// TIA Portal project "Palletizer" (V17)

(* hardware
DEVICE "S71500/ET200MP-Station_1"  S7-1500 station
   slot 0: "Profilschiene_0"  6ES7 590-1***0-0AA0
   slot 1: "PLC_1"  CPU 1511-1 PN  6ES7 511-1AK00-0AB0  V1.8
   slot 2: "AI 8xU/I/RTD/TC ST_1"  AI 8xU/I/RTD/TC ST  6ES7 531-7KF00-0AB0  V2.0
   slot 3: "AI 8xU/I/RTD/TC ST_2"  AI 8xU/I/RTD/TC ST  6ES7 531-7KF00-0AB0  V2.0
   slot 4: "AI 8xU/I/RTD/TC ST_3"  AI 8xU/I/RTD/TC ST  6ES7 531-7KF00-0AB0  V2.0
   slot 5: "AI 8xU/I/RTD/TC ST_4"  AI 8xU/I/RTD/TC ST  6ES7 531-7KF00-0AB0  V2.0
   slot 6: "DI 16x24VDC BA_1"  DI 16x24VDC BA  6ES7 521-1BH10-0AA0  V1.0
*)

// ===== PLC "PLC_1"  CPU 1511-1 PN =====

VAR_GLOBAL   // PLC tag table "Standard-Variablentabelle"
   "PALLET AT ENTRY" AT %E0.0 : Bool;
   "pallet at exit" AT %I0.1 : Bool;
   "pallet loaded" AT %I0.2 : Bool;
   "box at entry" AT %I0.3 : Bool;
   "pusher limit" AT %I0.4 : Bool;
   "plate limit" AT %I0.5 : Bool;
   "clamped" AT %I0.6 : Bool;
   "elevator moving" AT %I0.7 : Bool;
   "start" AT %I1.0 : Bool;
   "reset" AT %I1.1 : Bool;
   "stop" AT %I1.2 : Bool;
   "emergency stop" AT %I1.3 : Bool;
   "auto" AT %I1.4 : Bool;
   "factory run" AT %I1.5 : Bool;
   "pallet feeder" AT %Q0.0 : Bool;
   "load pallet" AT %Q0.1 : Bool;
   "exit conveyor" AT %Q0.2 : Bool;
   "move to limit" AT %Q0.3 : Bool;
   "elevator up" AT %Q0.4 : Bool;
   "elevator down" AT %Q0.5 : Bool;
   "box feeder" AT %Q0.6 : Bool;
   "turn" AT %Q0.7 : Bool;
   "push" AT %Q1.0 : Bool;
   "load belt" AT %Q1.1 : Bool;
   "clamp" AT %Q1.2 : Bool;
   "open plate" AT %Q1.3 : Bool;
   "warning light" AT %Q1.4 : Bool;
   "start light" AT %Q1.5 : Bool;
   "reset light" AT %Q1.6 : Bool;
   "stop light" AT %Q1.7 : Bool;
   "Tag_1" AT %M0.0 : Bool;
   "Tag_2" AT %M0.1 : Bool;
   "Tag_3" AT %M0.2 : Bool;
   "Tag_4" AT %M0.3 : Bool;
   "Tag_5" AT %M0.4 : Bool;
   "Tag_6" AT %M0.6 : Bool;
   "Tag_7" AT %M1.0 : Bool;
   "Tag_8" AT %MD100 : Time;
   "Tag_9" AT %M1.1 : Bool;
   "Tag_10" AT %MW100 : Int;
   "Tag_11" AT %M1.2 : Bool;
   "Tag_12" AT %M1.3 : Bool;
   "Tag_13" AT %MD200 : Time;
   "Tag_14" AT %M1.4 : Bool;
   "Tag_15" AT %M1.5 : Bool;
   "Tag_16" AT %MD300 : Time;
   "Tag_17" AT %M2.1 : Bool;
   "Tag_18" AT %M2.3 : Bool;
   "Tag_19" AT %M3.2 : Bool;
   "Tag_20" AT %M5.4 : Bool;
   "Tag_21" AT %M5.5 : Bool;
   "Tag_22" AT %M6.4 : Bool;
   "Tag_23" AT %M6.1 : Bool;
   "Tag_24" AT %M7.1 : Bool;
   "Tag_25" AT %M6.6 : Bool;
   "Tag_26" AT %M7.2 : Bool;
   "Tag_27" AT %M7.3 : Bool;
   "Tag_28" AT %M1.7 : Bool;
   "Tag_29" AT %M2.2 : Bool;
   "Tag_30" AT %M5.6 : Bool;
   "Tag_31" AT %M7.6 : Bool;
   "Tag_32" AT %M8.1 : Bool;
   "Tag_33" AT %M2.4 : Bool;
   "Tag_34" AT %M2.5 : Bool;
   "Tag_35" AT %M2.6 : Bool;
   "Tag_36" AT %M10.1 : Bool;
   "Tag_37" AT %MW400 : Int;
   "Tag_38" AT %QD30 : DWord;
END_VAR

// folder: System blocks/Program resources

DATA_BLOCK "IEC_Counter_0_DB"   // DB1
{ S7_Optimized_Access := 'TRUE' }
AUTHOR : Simatic
FAMILY : IEC
NAME : CNTR
VERSION : 1.0
// stored: InstanceOfName IEC_COUNTER
"IEC_COUNTER"
BEGIN
END_DATA_BLOCK

DATA_BLOCK "IEC_Timer_0_DB_1"   // DB2
{ S7_Optimized_Access := 'TRUE' }
AUTHOR : Simatic
FAMILY : IEC
NAME : IEC_TMR
VERSION : 1.0
// stored: InstanceOfName IEC_TIMER
"IEC_TIMER"
BEGIN
END_DATA_BLOCK

DATA_BLOCK "IEC_Timer_0_DB"   // DB3
{ S7_Optimized_Access := 'TRUE' }
AUTHOR : Simatic
FAMILY : IEC
NAME : IEC_TMR
VERSION : 1.0
// stored: InstanceOfName IEC_TIMER
"IEC_TIMER"
BEGIN
END_DATA_BLOCK

DATA_BLOCK "IEC_Counter_0_DB_1"   // DB4
{ S7_Optimized_Access := 'TRUE' }
AUTHOR : Simatic
FAMILY : IEC
NAME : CNTR
VERSION : 1.0
// stored: InstanceOfName IEC_COUNTER
"IEC_COUNTER"
BEGIN
END_DATA_BLOCK

DATA_BLOCK "IEC_Timer_0_DB_2"   // DB5
{ S7_Optimized_Access := 'TRUE' }
AUTHOR : Simatic
FAMILY : IEC
NAME : IEC_TMR
VERSION : 1.0
// stored: InstanceOfName IEC_TIMER
"IEC_TIMER"
BEGIN
END_DATA_BLOCK

DATA_BLOCK "IEC_Timer_0_DB_3"   // DB6
{ S7_Optimized_Access := 'TRUE' }
AUTHOR : Simatic
FAMILY : IEC
NAME : IEC_TMR
VERSION : 1.0
// stored: InstanceOfName IEC_TIMER
"IEC_TIMER"
BEGIN
END_DATA_BLOCK

DATA_BLOCK "IEC_Timer_0_DB_4"   // DB7
{ S7_Optimized_Access := 'TRUE' }
AUTHOR : Simatic
FAMILY : IEC
NAME : IEC_TMR
VERSION : 1.0
// stored: InstanceOfName IEC_TIMER
"IEC_TIMER"
BEGIN
END_DATA_BLOCK

DATA_BLOCK "IEC_Counter_0_DB_2"   // DB8
{ S7_Optimized_Access := 'TRUE' }
AUTHOR : Simatic
FAMILY : IEC
NAME : CNTR
VERSION : 1.0
// stored: InstanceOfName IEC_COUNTER
"IEC_COUNTER"
BEGIN
END_DATA_BLOCK

DATA_BLOCK "IEC_Timer_0_DB_5"   // DB9
{ S7_Optimized_Access := 'TRUE' }
AUTHOR : Simatic
FAMILY : IEC
NAME : IEC_TMR
VERSION : 1.0
// stored: InstanceOfName IEC_TIMER
"IEC_TIMER"
BEGIN
END_DATA_BLOCK

DATA_BLOCK "IEC_Timer_0_DB_6"   // DB10
{ S7_Optimized_Access := 'TRUE' }
AUTHOR : Simatic
FAMILY : IEC
NAME : IEC_TMR
VERSION : 1.0
// stored: InstanceOfName IEC_TIMER
"IEC_TIMER"
BEGIN
END_DATA_BLOCK

DATA_BLOCK "IEC_Timer_0_DB_7"   // DB11
{ S7_Optimized_Access := 'TRUE' }
AUTHOR : Simatic
FAMILY : IEC
NAME : IEC_TMR
VERSION : 1.0
// stored: InstanceOfName IEC_TIMER
"IEC_TIMER"
BEGIN
END_DATA_BLOCK

DATA_BLOCK "IEC_Timer_0_DB_8"   // DB12
{ S7_Optimized_Access := 'TRUE' }
AUTHOR : Simatic
FAMILY : IEC
NAME : IEC_TMR
VERSION : 1.0
// stored: InstanceOfName IEC_TIMER
"IEC_TIMER"
BEGIN
END_DATA_BLOCK

DATA_BLOCK "IEC_Timer_0_DB_9"   // DB13
{ S7_Optimized_Access := 'TRUE' }
AUTHOR : Simatic
FAMILY : IEC
NAME : IEC_TMR
VERSION : 1.0
// stored: InstanceOfName IEC_TIMER
"IEC_TIMER"
BEGIN
END_DATA_BLOCK

DATA_BLOCK "IEC_Counter_0_DB_3"   // DB14
{ S7_Optimized_Access := 'TRUE' }
AUTHOR : Simatic
FAMILY : IEC
NAME : CNTR
VERSION : 1.0
// stored: InstanceOfName IEC_COUNTER
"IEC_COUNTER"
BEGIN
END_DATA_BLOCK

DATA_BLOCK "IEC_Timer_0_DB_10"   // DB15
{ S7_Optimized_Access := 'TRUE' }
AUTHOR : Simatic
FAMILY : IEC
NAME : IEC_TMR
VERSION : 1.0
// stored: InstanceOfName IEC_TIMER
"IEC_TIMER"
BEGIN
END_DATA_BLOCK

DATA_BLOCK "IEC_Counter_0_DB_4"   // DB16
{ S7_Optimized_Access := 'TRUE' }
AUTHOR : Simatic
FAMILY : IEC
NAME : CNTR
VERSION : 1.0
// stored: InstanceOfName IEC_COUNTER
"IEC_COUNTER"
BEGIN
END_DATA_BLOCK

// folder: (top level)

FUNCTION "MHJ-PLC-Lab-Function-S71500" : Void   // FC9000, SCL
{ S7_Optimized_Access := 'TRUE' }
VERSION : 0.1
   VAR_TEMP
      Value : Byte;
      ForCounter : Int;
   END_VAR
   VAR CONSTANT
      Value_01_DW : DWord := 16#1223_5486;
      Value_02_DW : DWord := 16#A6C9_D1F5;
   END_VAR
BEGIN

   #Value:=PEEK(area := 16#82,
        dbNumber := 0,
        byteOffset := 511);
   #Value := #Value + 1;

   POKE(area := 16#82,
        dbNumber := 0,
        byteOffset := 511,
        value := #Value);

   POKE(area := 16#82,
        dbNumber := 0,
        byteOffset := 1016,
        value := #Value_01_DW);
   POKE(area := 16#82,
        dbNumber := 0,
        byteOffset := 1020,
        value := #Value_02_DW);

   FOR #ForCounter := 0 TO 63 DO
       #Value:=PEEK(area := 16#1,
            dbNumber := 0,
            byteOffset := #ForCounter);
       POKE(area := 16#81,
            dbNumber := 0,
            byteOffset := #ForCounter,
            value := #Value);
   END_FOR;
   #Value := PEEK(area := 16#1,
                  dbNumber := 0,
                  byteOffset := 512);
   POKE(area := 16#82,
        dbNumber := 0,
        byteOffset := 512,
        value := #Value);
END_FUNCTION

ORGANIZATION_BLOCK "Main"   // OB1, LAD, ProgramCycle
TITLE = "Main Program Sweep (Cycle)"
{ S7_Optimized_Access := 'TRUE' }
VERSION : 0.1
   VAR_INPUT
      Initial_Call : Bool;   // Initial call of this OB
      Remanence : Bool;   // =True, if remanent data are available
   END_VAR
   VAR_TEMP   // added for the SCL form of the ladder/FBD networks
      _w1 : Bool;
      _w2 : Bool;
   END_VAR
BEGIN

REGION Network 1
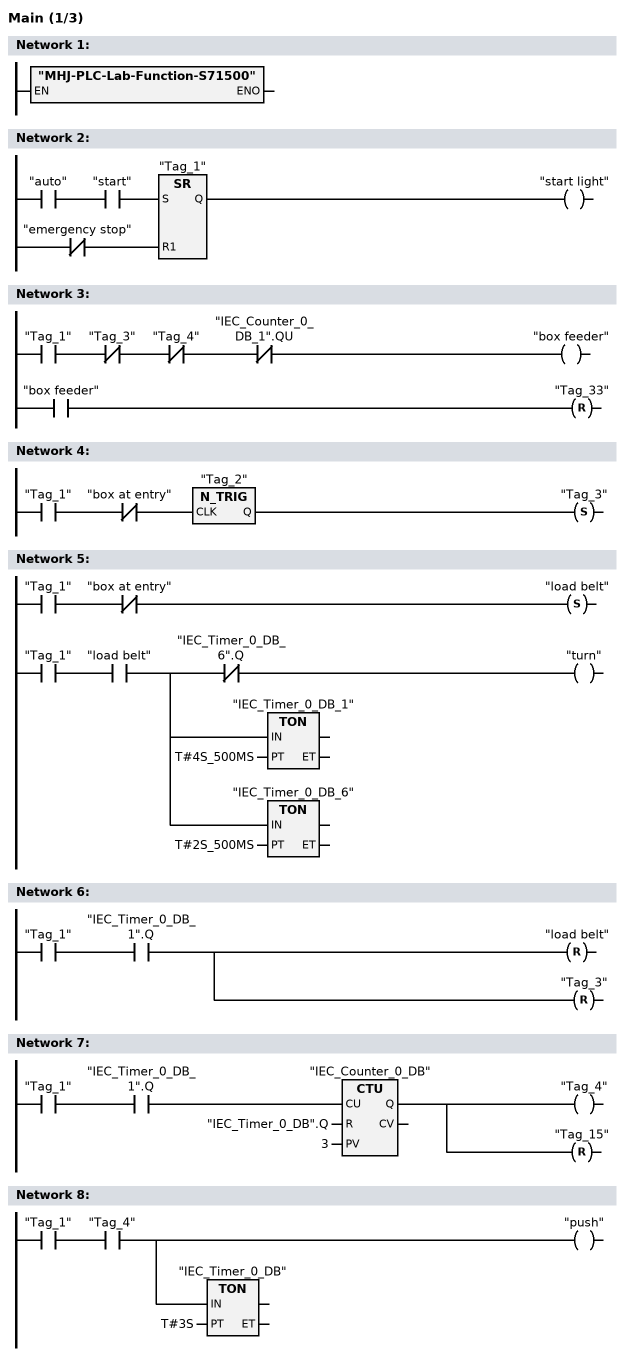
   RUNG wire#powerrail
      "MHJ-PLC-Lab-Function-S71500"()
   END_RUNG
   // the same network as SCL:
   "MHJ-PLC-Lab-Function-S71500"();
END_REGION

REGION Network 2
   RUNG wire#powerrail
      Contact( "auto" )
      Contact( "start" )
      S_SR(operand := "Tag_1", r1 := wire#w1)
      Coil( "start light" )
   END_RUNG
   RUNG wire#powerrail
      I_Contact( "emergency stop" )
   END_RUNG wire#w1
   // the same network as SCL:
   IF "auto" AND "start" THEN
       "Tag_1" := TRUE;   // SR flip-flop
   END_IF;
   IF NOT "emergency stop" THEN "Tag_1" := FALSE; END_IF;
   "start light" := "Tag_1";
END_REGION

REGION Network 3
   RUNG wire#powerrail
      Contact( "Tag_1" )
      I_Contact( "Tag_3" )
      I_Contact( "Tag_4" )
      I_Contact( "IEC_Counter_0_DB_1".QU )
      Coil( "box feeder" )
   END_RUNG
   RUNG wire#powerrail
      Contact( "box feeder" )
      R_Coil( "Tag_33" )
   END_RUNG
   // the same network as SCL:
   "box feeder" := "Tag_1" AND NOT "Tag_3" AND NOT "Tag_4" AND NOT "IEC_Counter_0_DB_1".QU;
   IF "box feeder" THEN "Tag_33" := FALSE; END_IF;
END_REGION

REGION Network 4
   RUNG wire#powerrail
      Contact( "Tag_1" )
      I_Contact( "box at entry" )
      N_Trig( "Tag_2" )
      S_Coil( "Tag_3" )
   END_RUNG
   // the same network as SCL:
   #_w1 := "Tag_1" AND NOT "box at entry";
   #_w2 := NOT #_w1 AND "Tag_2";   // falling edge
   "Tag_2" := #_w1;
   IF #_w2 THEN "Tag_3" := TRUE; END_IF;
END_REGION

REGION Network 5
   IF "Tag_1" AND NOT "box at entry" THEN "load belt" := TRUE; END_IF;
   #_w1 := "Tag_1" AND "load belt";
   "turn" := #_w1 AND NOT "IEC_Timer_0_DB_6".Q;
   "IEC_Timer_0_DB_1".TON(IN := #_w1, PT := T#4S_500MS);
   "IEC_Timer_0_DB_6".TON(IN := #_w1, PT := T#2S_500MS);
END_REGION

REGION Network 6
   RUNG wire#powerrail
      Contact( "Tag_1" )
      Contact( "IEC_Timer_0_DB_1".Q )
      wire#w1
      R_Coil( "load belt" )
   END_RUNG
   RUNG wire#w1
      R_Coil( "Tag_3" )
   END_RUNG
   // the same network as SCL:
   IF "Tag_1" AND "IEC_Timer_0_DB_1".Q THEN
       "load belt" := FALSE;
       "Tag_3" := FALSE;
   END_IF;
END_REGION

REGION Network 7
   "IEC_Counter_0_DB".CTU(CU := "Tag_1" AND "IEC_Timer_0_DB_1".Q, R := "IEC_Timer_0_DB".Q, PV := 3);
   "Tag_4" := "IEC_Counter_0_DB".Q;
   IF "IEC_Counter_0_DB".Q THEN "Tag_15" := FALSE; END_IF;
END_REGION

REGION Network 8
   "push" := "Tag_1" AND "Tag_4";
   "IEC_Timer_0_DB".TON(IN := "push", PT := T#3S);
END_REGION

REGION Network 9
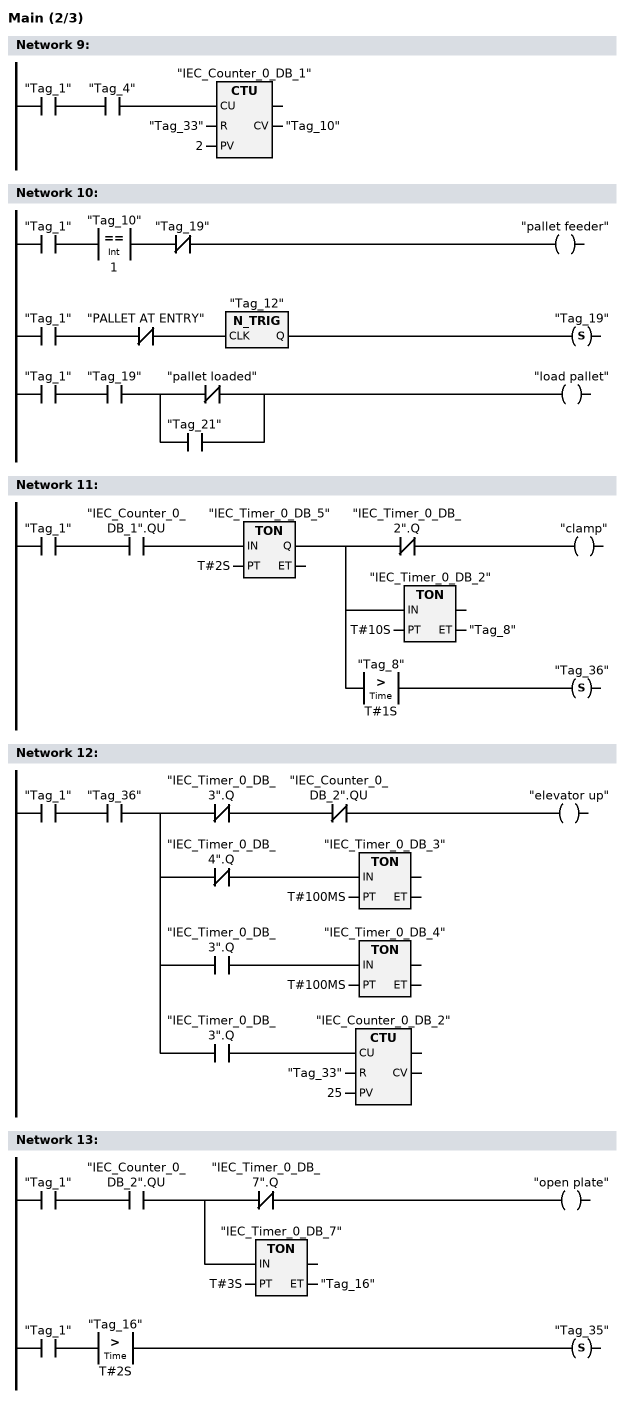
   "IEC_Counter_0_DB_1".CTU(CU := "Tag_1" AND "Tag_4", R := "Tag_33", PV := 2, CV => "Tag_10");
END_REGION

REGION Network 10
   RUNG wire#powerrail
      Contact( "Tag_1" )
      { S7_Templates := "SrcType := Int" } EQ_Contact(in1 := "Tag_10", in2 := 1)
      I_Contact( "Tag_19" )
      Coil( "pallet feeder" )
   END_RUNG
   RUNG wire#powerrail
      Contact( "Tag_1" )
      I_Contact( "PALLET AT ENTRY" )
      N_Trig( "Tag_12" )
      S_Coil( "Tag_19" )
   END_RUNG
   RUNG wire#powerrail
      Contact( "Tag_1" )
      Contact( "Tag_19" )
      wire#w1
      I_Contact( "pallet loaded" )
      wire#w2
      Coil( "load pallet" )
   END_RUNG
   RUNG wire#w1
      Contact( "Tag_21" )
   END_RUNG wire#w2
   // the same network as SCL:
   "pallet feeder" := "Tag_1" AND ("Tag_10" = 1) AND NOT "Tag_19";
   #_w1 := "Tag_1" AND NOT "PALLET AT ENTRY";
   #_w2 := NOT #_w1 AND "Tag_12";   // falling edge
   "Tag_12" := #_w1;
   IF #_w2 THEN "Tag_19" := TRUE; END_IF;
   "load pallet" := "Tag_1" AND "Tag_19" AND (NOT "pallet loaded" OR "Tag_21");
END_REGION

REGION Network 11
   "IEC_Timer_0_DB_5".TON(IN := "Tag_1" AND "IEC_Counter_0_DB_1".QU, PT := T#2S);
   "clamp" := "IEC_Timer_0_DB_5".Q AND NOT "IEC_Timer_0_DB_2".Q;
   "IEC_Timer_0_DB_2".TON(IN := "IEC_Timer_0_DB_5".Q, PT := T#10S, ET => "Tag_8");
   IF "IEC_Timer_0_DB_5".Q AND ("Tag_8" > T#1S) THEN "Tag_36" := TRUE; END_IF;
END_REGION

REGION Network 12
   #_w1 := "Tag_1" AND "Tag_36";
   "elevator up" := #_w1 AND NOT "IEC_Timer_0_DB_3".Q AND NOT "IEC_Counter_0_DB_2".QU;
   "IEC_Timer_0_DB_3".TON(IN := #_w1 AND NOT "IEC_Timer_0_DB_4".Q, PT := T#100MS);
   "IEC_Timer_0_DB_4".TON(IN := #_w1 AND "IEC_Timer_0_DB_3".Q, PT := T#100MS);
   "IEC_Counter_0_DB_2".CTU(CU := #_w1 AND "IEC_Timer_0_DB_3".Q, R := "Tag_33", PV := 25);
END_REGION

REGION Network 13
   #_w1 := "Tag_1" AND "IEC_Counter_0_DB_2".QU;
   "open plate" := #_w1 AND NOT "IEC_Timer_0_DB_7".Q;
   "IEC_Timer_0_DB_7".TON(IN := #_w1, PT := T#3S, ET => "Tag_16");
   IF "Tag_1" AND ("Tag_16" > T#2S) THEN "Tag_35" := TRUE; END_IF;
END_REGION

REGION Network 14
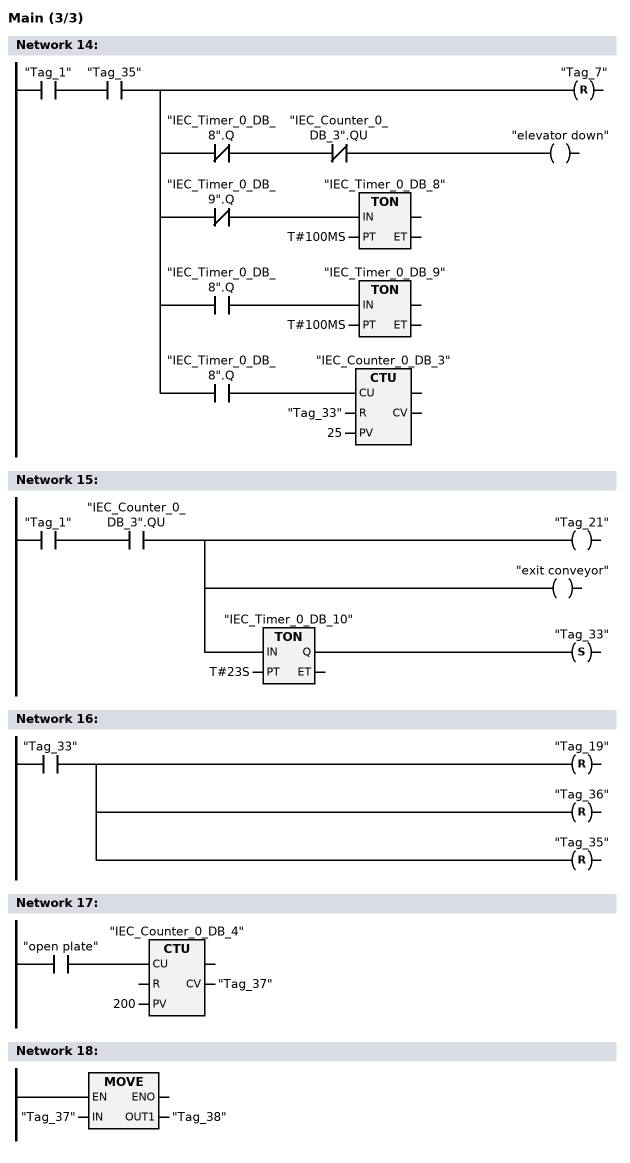
   #_w1 := "Tag_1" AND "Tag_35";
   IF #_w1 THEN "Tag_7" := FALSE; END_IF;
   "elevator down" := #_w1 AND NOT "IEC_Timer_0_DB_8".Q AND NOT "IEC_Counter_0_DB_3".QU;
   "IEC_Timer_0_DB_8".TON(IN := #_w1 AND NOT "IEC_Timer_0_DB_9".Q, PT := T#100MS);
   "IEC_Timer_0_DB_9".TON(IN := #_w1 AND "IEC_Timer_0_DB_8".Q, PT := T#100MS);
   "IEC_Counter_0_DB_3".CTU(CU := #_w1 AND "IEC_Timer_0_DB_8".Q, R := "Tag_33", PV := 25);
END_REGION

REGION Network 15
   "Tag_21" := "Tag_1" AND "IEC_Counter_0_DB_3".QU;
   "exit conveyor" := "Tag_21";
   "IEC_Timer_0_DB_10".TON(IN := "Tag_21", PT := T#23S);
   IF "IEC_Timer_0_DB_10".Q THEN "Tag_33" := TRUE; END_IF;
END_REGION

REGION Network 16
   RUNG wire#powerrail
      Contact( "Tag_33" )
      wire#w1
      R_Coil( "Tag_19" )
   END_RUNG
   RUNG wire#w1
      R_Coil( "Tag_36" )
   END_RUNG
   RUNG wire#w1
      R_Coil( "Tag_35" )
   END_RUNG
   // the same network as SCL:
   IF "Tag_33" THEN
       "Tag_19" := FALSE;
       "Tag_36" := FALSE;
       "Tag_35" := FALSE;
   END_IF;
END_REGION

REGION Network 17
   "IEC_Counter_0_DB_4".CTU(CU := "open plate", PV := 200, CV => "Tag_37");
END_REGION

REGION Network 18
   RUNG wire#powerrail
      Move(in := "Tag_37", out1 => "Tag_38")
   END_RUNG
   // the same network as SCL:
   "Tag_38" := "Tag_37";
END_REGION
END_ORGANIZATION_BLOCK